TYPE AxisIO :
STRUCT
	Enable		: BOOL;
END_STRUCT
END_TYPE

(* stored: Version 1.1.0.1, ProductVersion 3.1.4024.10
   DUT AxisIO: Id {b657be83-cdf7-43ac-b808-368fb04bf88d} *)
